{attribute 'hide'}
FUNCTION_BLOCK LongStringLen_Test EXTENDS TcUnit.FB_TestSuite

EmptyStringReturnsZero();
LongStringReturnsExpected();
ShortStringReturnsExpected();
T_MaxStringReturns255();

METHOD EmptyStringReturnsZero
VAR
	result : UDINT;
	value : STRING := '';
END_VAR
TEST('EmptyStringReturnsZero');

// @TEST-FIXTURE

// @TEST-RUN
result := LongStringLen(value);

// @TEST-ASSSERT
AssertEquals_UDINT(Expected := UDINT#0, Actual := result,
           Message := 'Empty string did not return zero');
		   

TEST_FINISHED();
END_METHOD

METHOD LongStringReturnsExpected
VAR
	result : UDINT;
	value : STRING(300) := '123456789012345678901234567890123456789012345678901234567890123456789012345678901234567890123456789012345678901234567890123456789012345678901234567890123456789012345678901234567890123456789012345678901234567890123456789012345678901234567890123456789012345678901234567890123456789012345678901234567890';
END_VAR
TEST('LongStringReturnsExpected');

// @TEST-FIXTURE

// @TEST-RUN
result := LongStringLen(value);

// @TEST-ASSSERT
AssertEquals_UDINT(Expected := UDINT#300, Actual := result,
           Message := 'Long string did not return expected');

TEST_FINISHED();
END_METHOD

METHOD ShortStringReturnsExpected
VAR
	result : UDINT;
	value : STRING := '1234567890';
END_VAR
TEST('ShortStringReturnsExpected');

// @TEST-FIXTURE

// @TEST-RUN
result := LongStringLen(value);

// @TEST-ASSSERT
AssertEquals_UDINT(Expected := UDINT#10, Actual := result,
           Message := 'Short string did not return expected');
		   

TEST_FINISHED();
END_METHOD

METHOD T_MaxStringReturns255
VAR
	result : UDINT;
	value : T_MaxString :='123456789012345678901234567890123456789012345678901234567890123456789012345678901234567890123456789012345678901234567890123456789012345678901234567890123456789012345678901234567890123456789012345678901234567890123456789012345678901234567890123456789012345';
END_VAR
TEST('T_MaxStringReturns255');

// @TEST-FIXTURE

// @TEST-RUN
result := LongStringLen(value);

// @TEST-ASSSERT
AssertEquals_UDINT(Expected := UDINT#255, Actual := result,
           Message := 'T_MaxString did not return 255');

TEST_FINISHED();
END_METHOD

END_FUNCTION_BLOCK

(* stored: Version 1.1.0.1, ProductVersion 3.1.4024.9
   POU LongStringLen_Test: Id {a705baa3-b0a7-47fe-9d51-8464a2b266cc}, SpecialFunc None
   Method EmptyStringReturnsZero: Id {aa7ed1ee-bd9f-4e2d-83f8-94d9ed5d9624}
   Method LongStringReturnsExpected: Id {da26980a-e645-4819-b21d-7c57cc917ffe}
   Method ShortStringReturnsExpected: Id {5978155d-bae8-457a-861d-4f461af82c52}
   Method T_MaxStringReturns255: Id {0a8a6a29-d0f3-407f-bd57-62b44af5b91b} *)
